{attribute 'GeneratedUsingTerminal: EL7411-0000-0016'}
{attribute addProperty BoxType "EL7411-0000-0016"}
{attribute addProperty Id "FB_PositionAT %I*FB_Position_3FA094ED4DRV_StatuswordAT %I*DRV_Statusword_9B36FDFC2DRV_Following_error_actual_valueAT %I*DRV_Following_error_actual_value_5AA320BF4DRV_ControlwordAT %Q*DRV_Controlword_F3F147212DRV_Target_positionAT %Q*DRV_Target_position_05240F144WcStateAT %I*WcState_9091E0EB2InfoDataAT %I*InfoData_6185D47C20"}
{attribute addProperty CRC "594204187"}
{attribute addProperty Size "38"}
TYPE EL7411_236AD61B EXTENDS EtcSlaveTerminalBase_947E5A46 :
STRUCT
	{attribute addProperty Name "FB_Position"}
	FB_Position : FB_Position_3FA094ED;
	{attribute addProperty Name "DRV_Statusword"}
	DRV_Statusword : DRV_Statusword_9B36FDFC;
	{attribute addProperty Name "DRV_Following_error_actual_value"}
	DRV_Following_error_actual_value : DRV_Following_error_actual_value_5AA320BF;
	{attribute addProperty Name "DRV_Controlword"}
	DRV_Controlword : DRV_Controlword_F3F14721;
	{attribute addProperty Name "DRV_Target_position"}
	DRV_Target_position : DRV_Target_position_05240F14;
	{attribute addProperty Name "WcState"}
	WcState : WcState_9091E0EB;
	{attribute addProperty Name "InfoData"}
	InfoData : InfoData_6185D47C;
END_STRUCT
END_TYPE

(* stored: Version 1.2.0.0, ProductVersion 3.1.4024.9
   DUT EL7411_236AD61B: Id {1a4dd9b2-0434-4aae-b7b1-57c658a03248} *)
